
// ===== library types =====

// folder: AWCModbus/Modbus Services

TYPE "typeMasterData"
VERSION : 0.1
   STRUCT
      Done : Bool;   // Request Completed
      Busy : Bool;   // Modbus Service is Busy
      Error : Bool;   // Request returned error
      locked : Bool;   // internal mutex **DO NOT WRITE TO**
      Mode : USInt;   // internal mode **DO NOTE WRITE TO**
      Status : Int;   // Request Status
      "Slave ID" : UInt;   // internal slave ID **DO NOTE WRITE TO**
      "Register Address" : UDInt;   // internal register address **DO NOTE WRITE TO**
      Length : UInt;   // internal length **DO NOTE WRITE TO**
      RequestID : UInt;   // Request ID **DO NOTE WRITE TO**
      Data : Array[0..299] of Byte;   // Returned Data **DO NOTE WRITE TO**
   END_STRUCT;
END_TYPE

// folder: AWCModbus/01_Modbus Services

FUNCTION_BLOCK "ModbusRtuEngine"   // FB6, LAD
TITLE = ModbusRTUEngine
{ S7_Optimized_Access := 'TRUE' }
AUTHOR : Matt_Paulissen
FAMILY : AWCModbus
NAME : ModbusRTUEngine
// Modbus polling service for RTU devices.
   VAR_INPUT
      port : Port;   // The port references the “HW_Address” of the interface that will be used for Modbus communication. In the above example the “Local~CB_1241_(RS485) is referenced.
      baudRate : UDInt;   // The baud rate determines the communications speed of the network. All devices on the network must be set to the same baud rate. Available options are: 300, 600, 1200, 2400, 4800, 9600, 19200, 38400, 57600, 76800, 115200 bit/s.
      parity : UInt;   // Used to set the network parity. All devices on the network must have the same parity setting. Available options are: 0 = None, 1 = Odd, 2= Even.
      FirstScan : Bool;   // First Scan is used to initialize the communications port on system start up. This input can also be used at other times if it is desired to reset the communications parameters without restarting the CPU.
      Reset : Bool;   // Used to reinitialize the communications port of the CPU or module.
   END_VAR
   VAR_OUTPUT
      Status : Int;   // Returns any error code for the Modus Master function.
   END_VAR
   VAR_IN_OUT
      masterInterface : "typeMasterData";   // The “Master Interface” parameter is used to pass date between the Modbus RTU Engine and subsequent read and write function. The data type is the user defined type “typeMasterData”. It is necessary to create a global data block containing one instance of the “typeMasterData”.
   END_VAR
   VAR
      statPrevious : Int;
      statCurrent : Int;
      statIndex : Int;
      statRequestID : UInt;
      Comm_Load_Status : Int;
      Comm_Load_Done : Bool;
      Comm_Load_Error : Bool;
      instStuckInterfaceTimer : TON_TIME;
      instReinitilizeTimer : TON_TIME;
      instCommLoad : Modbus_Comm_Load;
      instMaster : Modbus_Master;
      inst7002Timeout : TON_TIME;
   END_VAR
   VAR_TEMP
      tempServerStatus : Int;
   END_VAR
   VAR CONSTANT
      UNITIALIZED : Int := 0;
      INITIALIZING_PORT : Int := 1;
      POLLING : Int := 2;
      POLLING_DONE : Int := 3;
   END_VAR
   VAR_TEMP   // added for the SCL form of the ladder/FBD networks
      _w1 : Bool;
   END_VAR
BEGIN

REGION Network 1: BLOCK INFO HEADER
   // AWC INC / (c)Copyright 2022
   // ------------------------------------------------------------------------------
   // Title:            ModbusRTUEngine_xxx
   // Comment/Function: Modbus Polling Service for RTU Devices:
   // Library/Family:   AWCModbus
   // Author:           Matt Paulissen
   // Tested with:      ---
   // Engineering:      TIA Portal V17
   // Restrictions:     -
   // Requirements:     ---
   // ------------------------------------------------------------------------------
   // Change log table:
   // Version  | Date       | Expert in charge       | Changes applied
   // ---------|------------|------------------------|------------------------------
   // 01.00.00 | 06.18.2018 | F.Maynard, M.Paulissen
   //                                Initial Release
   // 01.01.00 | 01.25.2019 | F.Maynard, M.Paulissen
   //                                Changed to RTU block that works for 1500 as well as 1200.
   // 02.00.00 | 03.12.2019 | F.Maynard, M.Paulissen
   //                                Changed all blocks to Optimized data access and added software unit.
   // 02.01.00 | 09.01.2019 | F.Maynard, M.Paulissen
   //                                Updated RTU engine to V4.3 instructions
   // 02.02.00 | 09.25.2019 | F.Maynard, M.Paulissen
   //                                Added remote TCP port for the TCP engine
   // 02.03.00 | 10.14.2019 | F.Maynard, M.Paulissen
   //                                 Bugfix for CM_PTP lockup
END_REGION

REGION Network 2: DESCRIPTION
   // The “ModbusRTUEngine” is used to communicate via Modbus RTU via an RS-485, RS-422, or RS-232 communications add on module.  The parameters are used to initialize the communication port, set the baud rate, and parity.
   // 
   // ---
   // 
   // CAUTION
   // :    You must change the mode parameter in instCommLoad to the correct value for your serial module
   // 
   // ---
END_REGION

REGION Network 3: Run Comm Load
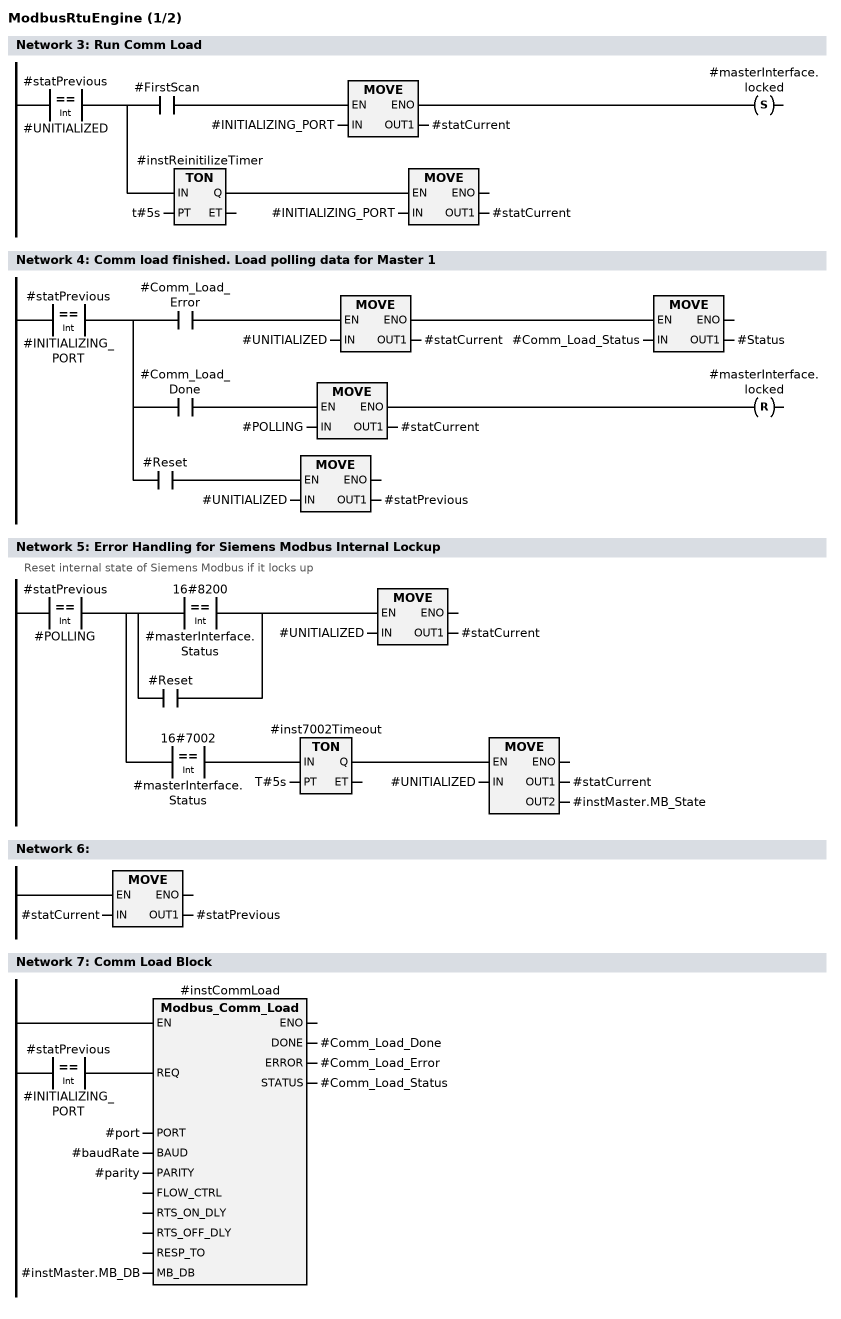
   #_w1 := #statPrevious = #UNITIALIZED;
   IF #_w1 AND #FirstScan THEN
       #statCurrent := #INITIALIZING_PORT;
       #masterInterface.locked := TRUE;
   END_IF;
   #instReinitilizeTimer(IN := #_w1, PT := t#5s);   // TON
   IF #instReinitilizeTimer.Q THEN #statCurrent := #INITIALIZING_PORT; END_IF;
END_REGION

REGION Network 4: Comm load finished. Load polling data for Master 1
   RUNG wire#powerrail
      { S7_Templates := "SrcType := Int" } EQ_Contact(in1 := #statPrevious, in2 := #INITIALIZING_PORT)
      wire#w1
      Contact( #Comm_Load_Error )
      Move(in := #UNITIALIZED, out1 => #statCurrent)
      Move(in := #Comm_Load_Status, out1 => #Status)
   END_RUNG
   RUNG wire#w1
      Contact( #Comm_Load_Done )
      Move(in := #POLLING, out1 => #statCurrent)
      R_Coil( #masterInterface.locked )
   END_RUNG
   RUNG wire#w1
      Contact( #Reset )
      Move(in := #UNITIALIZED, out1 => #statPrevious)
   END_RUNG
   // the same network as SCL:
   #_w1 := #statPrevious = #INITIALIZING_PORT;
   IF #_w1 AND #Comm_Load_Error THEN
       #statCurrent := #UNITIALIZED;
       #Status := #Comm_Load_Status;
   END_IF;
   IF #_w1 AND #Comm_Load_Done THEN
       #statCurrent := #POLLING;
       #masterInterface.locked := FALSE;
   END_IF;
   IF #_w1 AND #Reset THEN #statPrevious := #UNITIALIZED; END_IF;
END_REGION

REGION Network 5: Error Handling for Siemens Modbus Internal Lockup
   // Reset internal state of Siemens Modbus if it locks up
   #_w1 := #statPrevious = #POLLING;
   IF #_w1 AND ((16#8200 = #masterInterface.Status) OR #Reset) THEN #statCurrent := #UNITIALIZED; END_IF;
   #inst7002Timeout(IN := #_w1 AND (16#7002 = #masterInterface.Status), PT := T#5s);   // TON
   IF #inst7002Timeout.Q THEN
       #statCurrent := #UNITIALIZED;
       #instMaster.MB_State := #UNITIALIZED;
   END_IF;
END_REGION

REGION Network 6
   RUNG wire#powerrail
      Move(in := #statCurrent, out1 => #statPrevious)
   END_RUNG
   // the same network as SCL:
   #statPrevious := #statCurrent;
END_REGION

REGION Network 7: Comm Load Block
   #instCommLoad(REQ := #statPrevious = #INITIALIZING_PORT,   // Modbus_Comm_Load
                 PORT := #port,
                 BAUD := #baudRate,
                 PARITY := #parity,
                 MB_DB := #instMaster.MB_DB,
                 DONE => #Comm_Load_Done,
                 ERROR => #Comm_Load_Error,
                 STATUS => #Comm_Load_Status);
END_REGION

REGION Network 8: Master Instance 1
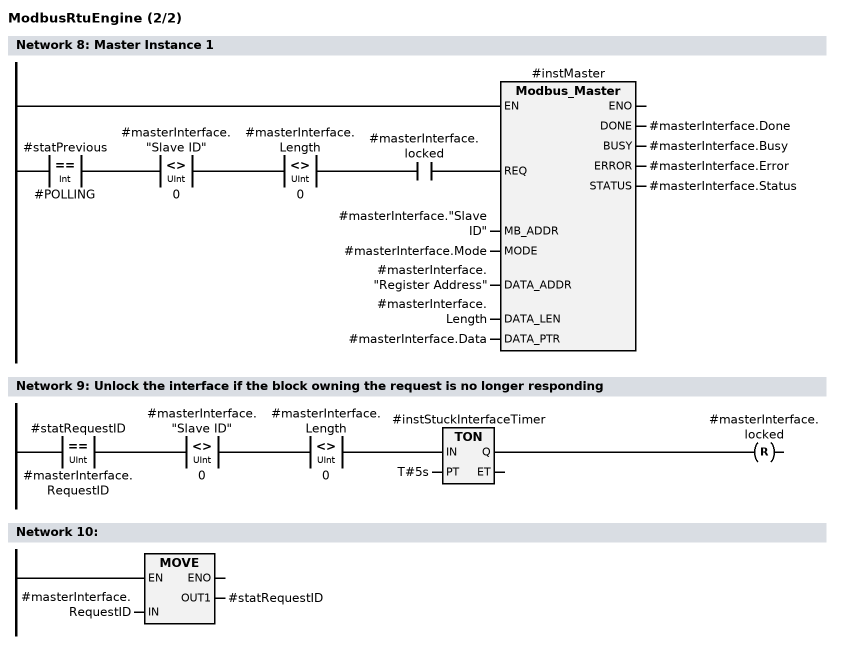
   #instMaster(REQ := (#statPrevious = #POLLING) AND (#masterInterface."Slave ID" <> 0) AND (#masterInterface.Length <> 0) AND #masterInterface.locked,   // Modbus_Master
               MB_ADDR := #masterInterface."Slave ID",
               MODE := #masterInterface.Mode,
               DATA_ADDR := #masterInterface."Register Address",
               DATA_LEN := #masterInterface.Length,
               DATA_PTR := #masterInterface.Data,
               DONE => #masterInterface.Done,
               BUSY => #masterInterface.Busy,
               ERROR => #masterInterface.Error,
               STATUS => #masterInterface.Status);
END_REGION

REGION Network 9: Unlock the interface if the block owning the request is no longer responding
   #instStuckInterfaceTimer(IN := (#statRequestID = #masterInterface.RequestID) AND (#masterInterface."Slave ID" <> 0) AND (#masterInterface.Length <> 0),   // TON
                           PT := T#5s);
   IF #instStuckInterfaceTimer.Q THEN #masterInterface.locked := FALSE; END_IF;
END_REGION

REGION Network 10
   RUNG wire#powerrail
      Move(in := #masterInterface.RequestID, out1 => #statRequestID)
   END_RUNG
   // the same network as SCL:
   #statRequestID := #masterInterface.RequestID;
END_REGION
END_FUNCTION_BLOCK

FUNCTION_BLOCK "ModbusTCPEngine"   // FB22, LAD
TITLE = ModbusTCPEngine
{ S7_Optimized_Access := 'TRUE' }
AUTHOR : Matt_Paulissen
FAMILY : AWCModbus
NAME : ModbusTCPEngine
VERSION : 0.1
// The “ModbusTCPEngine” is used to communicate via Modbus TCP via the on-board Profinet port or via a separate add on Ethernet communications module.
   VAR_INPUT
      port : Hw_Any;   // The port references the “HW_Address” of the Profinet interface that will be used for Modbus TCP communication. In the above example the “Local~Profinet_interface_1” is referenced.
      connectionId : Conn_Ouc;   // Defines the unique connection id for the Modbus Client. If more than one instance of the Modbus Client is used a different connection id must be assigned.
      tcpPort : UInt;   // Modbus TCP Server TCP Port Number. Typically this is port 502, but in some instances may be changed to meet network requirements.
      ipOne : Byte;   // First address octet of the server to be polled.
      ipTwo : Byte;   // Second address octet of the server to be polled.
      ipThree : Byte;   // Third address octet of the server to be polled.
      ipFour : Byte;   // Fourth address octet of the server to be polled.
   END_VAR
   VAR_OUTPUT
      Status : Int;   // Returns any error code for the Modbus Client function.
   END_VAR
   VAR_IN_OUT
      masterInterface : "typeMasterData";   // The “Master Interface” parameter is used to pass date between the Modbus RTU Engine and subsequent read and write function. The data type is the user defined type “typeMasterData”. It is necessary to create a global data block containing one instance of the “typeMasterData”.
   END_VAR
   VAR
      instClient : MB_CLIENT;
      connection : TCON_IP_v4;
      statRequestID : UInt;
      instStuckInterfaceTimer : TON_TIME;
   END_VAR
   VAR CONSTANT
      UNITIALIZED : Int := 0;
      INITIALIZING_PORT : Int := 1;
      POLLING_ONE : Int := 2;
      POLLING_DONE_ONE : Int := 3;
      POLLING_TWO : Int := 4;
      POLLING_TWO_DONE : Int := 5;
   END_VAR
   // connection.ConnectionType := 11;
   // connection.ActiveEstablished := 1;
   // connection.RemotePort := 502;
   // connection.LocalPort := 502;
BEGIN

REGION Network 1: BLOCK INFO HEADER
   // AWC INC / (c)Copyright 2022
   // ------------------------------------------------------------------------------
   // Title:            ModbusTCPEngine_xxx
   // Comment/Function: Modbus Polling Service for RTU Devices:
   // Library/Family:   AWCModbus
   // Author:           Matt Paulissen
   // Tested with:      ---
   // Engineering:      TIA Portal V17
   // Restrictions:     -
   // Requirements:     ---
   // ------------------------------------------------------------------------------
   // Change log table:
   // Version  | Date       | Expert in charge       | Changes applied
   // ---------|------------|------------------------|------------------------------
   // 01.00.00 | 06.18.2018 | F.Maynard, M.Paulissen | Initial Release
   // 01.01.00 | 01.25.2019 | F.Maynard, M.Paulissen | Changed to RTU block that works for 1500 as well as 1200.  Added Devices folder for common devices.  Added ability to read from contacts and write to coils with Boolean tags
   // 02.00.00 | 03.12.2019 | F.Maynard, M.Paulissen | Changed all blocks to Optimized data access and added software unit.
   // 02.01.00 | 09.01.2019 | F.Maynard, M.Paulissen | Updated RTU engine to V4.3 instructions
   // 02.02.00 | 09.25.2019 | F.Maynard, M.Paulissen | Added remote TCP port for the TCP engine
   // 02.03.00 | 10.14.2019 | F.Maynard, M.Paulissen | Bugfix for CM_PTP lockup
END_REGION

REGION Network 2: DESCRIPTION
   // The “ModbusTCPEngine” is used to communicate via Modbus TCP via the on-board Profinet port or via a separate add on Ethernet communications module.
END_REGION

REGION Network 3: Move ip address from interface to static tcon_ip_v4
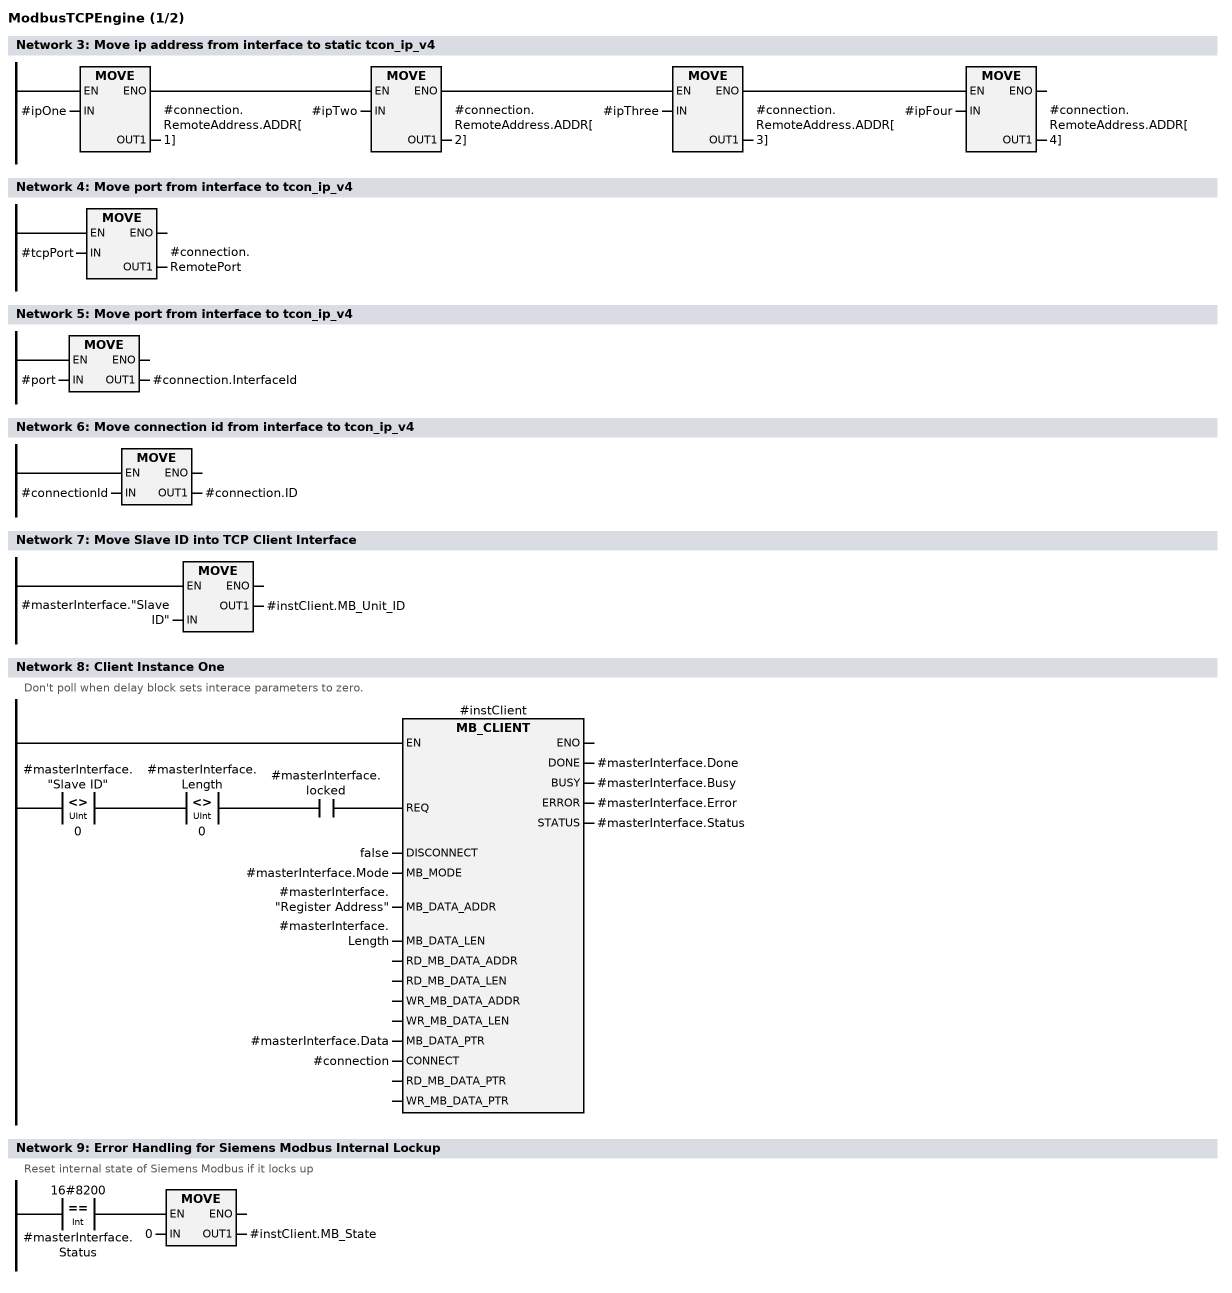
   RUNG wire#powerrail
      Move(in := #ipOne, out1 => #connection.RemoteAddress.ADDR[1])
      Move(in := #ipTwo, out1 => #connection.RemoteAddress.ADDR[2])
      Move(in := #ipThree, out1 => #connection.RemoteAddress.ADDR[3])
      Move(in := #ipFour, out1 => #connection.RemoteAddress.ADDR[4])
   END_RUNG
   // the same network as SCL:
   #connection.RemoteAddress.ADDR[1] := #ipOne;
   #connection.RemoteAddress.ADDR[2] := #ipTwo;
   #connection.RemoteAddress.ADDR[3] := #ipThree;
   #connection.RemoteAddress.ADDR[4] := #ipFour;
END_REGION

REGION Network 4: Move port from interface to tcon_ip_v4
   RUNG wire#powerrail
      Move(in := #tcpPort, out1 => #connection.RemotePort)
   END_RUNG
   // the same network as SCL:
   #connection.RemotePort := #tcpPort;
END_REGION

REGION Network 5: Move port from interface to tcon_ip_v4
   RUNG wire#powerrail
      Move(in := #port, out1 => #connection.InterfaceId)
   END_RUNG
   // the same network as SCL:
   #connection.InterfaceId := #port;
END_REGION

REGION Network 6: Move connection id from interface to tcon_ip_v4
   RUNG wire#powerrail
      Move(in := #connectionId, out1 => #connection.ID)
   END_RUNG
   // the same network as SCL:
   #connection.ID := #connectionId;
END_REGION

REGION Network 7: Move Slave ID into TCP Client Interface
   RUNG wire#powerrail
      Move(in := #masterInterface."Slave ID", out1 => #instClient.MB_Unit_ID)
   END_RUNG
   // the same network as SCL:
   #instClient.MB_Unit_ID := #masterInterface."Slave ID";
END_REGION

REGION Network 8: Client Instance One
   // Don't poll when delay block sets interace parameters to zero.
   #instClient(REQ := (#masterInterface."Slave ID" <> 0) AND (#masterInterface.Length <> 0) AND #masterInterface.locked,   // MB_CLIENT
               DISCONNECT := false,
               MB_MODE := #masterInterface.Mode,
               MB_DATA_ADDR := #masterInterface."Register Address",
               MB_DATA_LEN := #masterInterface.Length,
               MB_DATA_PTR := #masterInterface.Data,
               CONNECT := #connection,
               DONE => #masterInterface.Done,
               BUSY => #masterInterface.Busy,
               ERROR => #masterInterface.Error,
               STATUS => #masterInterface.Status);
END_REGION

REGION Network 9: Error Handling for Siemens Modbus Internal Lockup
   // Reset internal state of Siemens Modbus if it locks up
   RUNG wire#powerrail
      { S7_Templates := "SrcType := Int" } EQ_Contact(in1 := 16#8200, in2 := #masterInterface.Status)
      Move(in := 0, out1 => #instClient.MB_State)
   END_RUNG
   // the same network as SCL:
   IF 16#8200 = #masterInterface.Status THEN #instClient.MB_State := 0; END_IF;
END_REGION

REGION Network 10: Unlock the interface if the block owning the request is no longer responding
   // Modbus Polling Delay block sets interfaces to zero.  Don't want to unlock interface if this block is holding it.
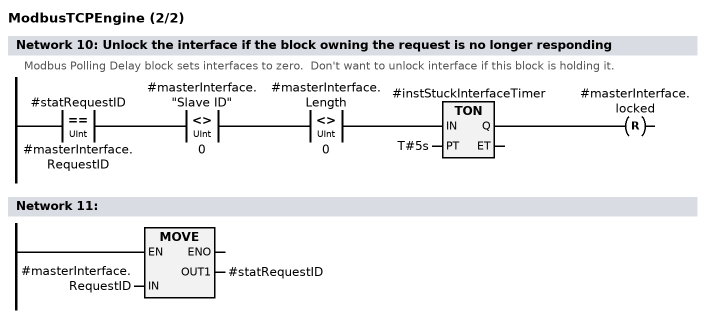
   #instStuckInterfaceTimer(IN := (#statRequestID = #masterInterface.RequestID) AND (#masterInterface."Slave ID" <> 0) AND (#masterInterface.Length <> 0),   // TON
                           PT := T#5s);
   IF #instStuckInterfaceTimer.Q THEN #masterInterface.locked := FALSE; END_IF;
END_REGION

REGION Network 11
   RUNG wire#powerrail
      Move(in := #masterInterface.RequestID, out1 => #statRequestID)
   END_RUNG
   // the same network as SCL:
   #statRequestID := #masterInterface.RequestID;
END_REGION
END_FUNCTION_BLOCK

// folder: AWCModbus/01_Modbus Services/Modbus Polling Functions

FUNCTION "GeneralModbusPoll" : Void   // FC11, SCL
TITLE = GeneralModbusPoll
{ S7_Optimized_Access := 'TRUE' }
AUTHOR : Matt_Paulissen
FAMILY : AWCModbus
NAME : GeneralModbusPoll
VERSION : 0.1
// The General Modbus Poll Function is used to read a single data value from the Modbus RTU slave or Modbus TCP server.
   VAR_INPUT
      slaveId : Int;   // When using the function for Modbus RTU this will be the remote slave network address. When using the function for Modbus TCP this will be the device address, in most instances this value will be 1, unless there is a Modbus TCP to Modbus RTU gateway employed. If there is a Modbus TCP to Modbus RTU gateway this value will point to the slave device address on the Modbus RTU side of the gateway.
      address : UDInt;   // The address parameter references the Modbus register that will be polled.
      swappedFloatingPoint : Bool;   // When reading floating point values from some devices it is necessary to reverse the order of the received data words to display the value correctly. In this it is necessary to set this value to True.
      substituteValue : Real;   // If the remote device fails to respond or has an error the Substitute Value will be returned to the Data value. This can be used to alert the operator that there is a problem with the connection.
   END_VAR
   VAR_OUTPUT
      data : Variant;   // The Data parameter is the value returned from the device. The data type of the PLC variable selected will determine how many registers are requested from the device and how they are displayed in the PLC.
   END_VAR
   VAR_IN_OUT
      modbusInterface : "typeMasterData";   // The “Master Interface” parameter is used to pass date between the Modbus RTU Engine and subsequent read and write function. The data type is the user defined type “typeMasterData”. It is necessary to create a global data block containing one instance of the “typeMasterData”.
   END_VAR
   VAR_TEMP
      tempArray : Array[0..3] of Byte;
      tempDWord : DWord;
      tempStatus : Int;
      tempPos : DInt;
      tempBool : Bool;
   END_VAR
BEGIN
   REGION BLOCK INFO HEADER
       //===============================================================================
       // AWC INC / (c)Copyright 2022
       //-------------------------------------------------------------------------------
       // Title:            GeneralModbusPoll_xxx
       // Comment/Function: Poll an individual value from a Modbus Device
       // Library/Family:   AWCModbus
       // Author:           Matt Paulissen
       // Tested with:      ---
       // Engineering:      TIA Portal V17
       // Restrictions:     ---
       // Requirements:     ---
       //-------------------------------------------------------------------------------
       // Change log table:
       // Version  | Date       | Expert in charge       | Changes applied
       //----------|------------|------------------------|------------------------------
       // 01.00.00 | 08.09.2017 | Matt Paulissen | First released version
       // 01.00.01 | 08.23.2017 | Matt Paulissen | Added ability to set failover value
       // 01.00.02 | 09.21.2018 | Matt Paulissen | Added request ID to detect stuck lock
       // 01.01.00 | 01.25.2019 | Matt Paulissen | Added ability to read contacts
       // 01.01.01 | 11.04.2022 | Matt Paulissen | Bug fix for substitute value on DWord
       //===============================================================================
   END_REGION

   REGION DESCRIPTION
       (/*The General Modbus Poll Function is used to read a single data value from the Modbus RTU slave or Modbus TCP server.*/)
   END_REGION DESCRIPTION

   //Check for lock
   IF (NOT #modbusInterface.locked) THEN
       //Move Register and Slave address to Modbus Register
       #modbusInterface."Slave ID" := #slaveId;
       #modbusInterface."Register Address" := #address;
       #modbusInterface.Mode := 0;
       CASE TypeOf(#data) OF
           UInt:
               #modbusInterface.Length := 1;
           Int:
               #modbusInterface.Length := 1;
           Word:
               #modbusInterface.Length := 1;
           DWord:
               #modbusInterface.Length := 2;
           Real:
               #modbusInterface.Length := 2;
           Bool:
               #modbusInterface.Length := 1;
           ELSE  // Statement section ELSE
               ;
       END_CASE;
       #modbusInterface.locked := TRUE;
       #modbusInterface.RequestID += 1;
       RETURN;
   END_IF;
   IF ((#modbusInterface.locked)
       AND (
       (#modbusInterface."Slave ID" = #slaveId)
       AND (#modbusInterface."Register Address" = #address)
       AND (#modbusInterface.Mode = 0))
       )
   THEN
       IF (#modbusInterface.Done) THEN
           //Inspect type of output and set correct type of input in modbus register
           CASE TypeOf(#data) OF
               UInt:
                   #tempStatus := Deserialize(SRC_ARRAY := #modbusInterface.Data,
                                              DEST_VARIABLE => #data,
                                              POS := #tempPos);
               Int:
                   #tempStatus := Deserialize(SRC_ARRAY := #modbusInterface.Data,
                                              DEST_VARIABLE => #data,
                                              POS := #tempPos);
               Word:
                   #tempStatus := Deserialize(SRC_ARRAY := #modbusInterface.Data,
                                              DEST_VARIABLE => #data,
                                              POS := #tempPos);
               DWord:
                   IF #swappedFloatingPoint THEN
                       // Swapped 
                       #tempArray[3] := #modbusInterface.Data[1];
                       #tempArray[2] := #modbusInterface.Data[0];
                       #tempArray[1] := #modbusInterface.Data[3];
                       #tempArray[0] := #modbusInterface.Data[2];
                       #tempStatus := Deserialize(SRC_ARRAY := #tempArray,
                                                  DEST_VARIABLE => #data,
                                                  POS := #tempPos);
                   ELSE
                       //Consecutive
                       #tempStatus := Deserialize(SRC_ARRAY := #modbusInterface.Data,
                                                  DEST_VARIABLE => #data,
                                                  POS := #tempPos);
                   END_IF;

               Real:
                   IF #swappedFloatingPoint THEN
                       // Swapped 
                       #tempArray[3] := #modbusInterface.Data[1];
                       #tempArray[2] := #modbusInterface.Data[0];
                       #tempArray[1] := #modbusInterface.Data[3];
                       #tempArray[0] := #modbusInterface.Data[2];
                       #tempStatus := Deserialize(SRC_ARRAY := #tempArray,
                                                  DEST_VARIABLE => #data,
                                                  POS := #tempPos);

                   ELSE
                       //Consecutive
                       #tempStatus := Deserialize(SRC_ARRAY := #modbusInterface.Data,
                                                  DEST_VARIABLE => #data,
                                                  POS := #tempPos);
                   END_IF;

               Bool:
                   #tempBool := #modbusInterface.Data[0].%X0;
                   VariantPut(SRC := #tempBool,
                              DST := #data);
               ELSE  // Statement section ELSE
                   ;
           END_CASE;
           #modbusInterface.locked := FALSE;
       END_IF;
       IF (#modbusInterface.Error) THEN
           CASE TypeOf(#data) OF
               UInt:
                   VariantPut(SRC := REAL_TO_UINT(IN:=#substituteValue),
                              DST := #data);
               Int:
                   VariantPut(SRC := REAL_TO_INT(IN := #substituteValue),
                              DST := #data);
               Word:
                   VariantPut(SRC := INT_TO_WORD(IN:=TRUNC_INT(IN := #substituteValue)),
                              DST := #data);
               DWord:
                   VariantPut(SRC := REAL_TO_DWORD(IN:=#substituteValue),
                              DST := #data);
               Real:
                   VariantPut(SRC := #substituteValue,
                              DST := #data);
               Bool:
                   IF (#substituteValue <> 0.0) THEN
                       #tempBool := TRUE;
                   ELSE
                       #tempBool := FALSE;
                   END_IF;
                   VariantPut(SRC := #tempBool,
                              DST := #data);
               ELSE  // Statement section ELSE
                   ;
           END_CASE;
           #modbusInterface.locked := 0;
       END_IF;
   END_IF;
END_FUNCTION

FUNCTION "LargeModbusPoll" : Void   // FC892, SCL
TITLE = LargeModbusPoll
{ S7_Optimized_Access := 'TRUE' }
AUTHOR : Matt_Paulissen
FAMILY : AWCModbus
NAME : LargeModbusPoll
VERSION : 0.1
// Large Modbus Poll function is used to read multiple contiguous data values from a Modbus RTU slave or Modbus TCP Server. Number of values read is determined by the size of the Array element at the Data parameter.
   VAR_INPUT
      slaveId : Int;   // When using the function for Modbus RTU this will be the remote slave network address. When using the function for Modbus TCP this will be the device address, in most instances this value will be 1, unless there is a Modbus TCP to Modbus RTU gateway employed. If there is a Modbus TCP to Modbus RTU gateway this value will point to the slave device address on the Modbus RTU side of the gateway.
      address : UDInt;   // The address parameter references the Modbus register that will be polled.
   END_VAR
   VAR_OUTPUT
      data : Variant;   // The Data parameter is the value returned from the device. The data type of the PLC variable selected will determine how many registers are requested from the device and how they are displayed in the PLC. The allowable data types are: Int, UInt, Word, Dint, UDint, DWord, and Real, Array of Uint, Array of Int, Array of Udint, Array of Dint, Array of Real, and PLC UDTs. Care should be taken to not exceed the 127-byte limitation of the Modbus Read Function.
      status : Int;   // Returns any error code for the Modbus Master function.
   END_VAR
   VAR_IN_OUT
      modbusInterface : "typeMasterData";   // The “Master Interface” parameter is used to pass datae between the Modbus RTU Engine and subsequent read and write function. The data type is the user defined type “typeMasterData”. It is necessary to create a global data block containing one instance of the “typeMasterData”.
   END_VAR
   VAR_TEMP
      tempPosition : DInt;
      tempStatus : Int;
      tempMode : USInt;
      tempAddress : UInt;
   END_VAR
BEGIN
   REGION BLOCK INFO HEADER
       //===============================================================================
       // AWC INC / (c)Copyright 2022
       //-------------------------------------------------------------------------------
       // Title:            LargeModbusPoll_xxx
       // Comment/Function: Read multiple contiguous values from a Modbus Device
       // Library/Family:   AWCModbus
       // Author:           Matt Paulissen
       // Tested with:      ---
       // Engineering:      TIA Portal V17
       // Restrictions:     ---
       // Requirements:     ---
       //-------------------------------------------------------------------------------
       // Change log table:
       // Version  | Date       | Expert in charge       | Changes applied
       //----------|------------|------------------------|------------------------------
       // 01.00.00 | 05.17.2018 | Matt Paulissen | First released version
       // 01.00.02 | 09.21.2018 | Matt Paulissen | Added request ID to detect stuck lock
       // 01.01.06 | 09.29.2020 | Matt Paulissen | Added extended modbus addressing
       // 01.01.07 | 11.16.2022 | Matt Paulissen | Allowed UDint for addresses
       //===============================================================================
   END_REGION

   REGION DESCRIPTION
       (/*Large Modbus Poll function is used to read multiple contiguous data values from a Modbus RTU slave or Modbus TCP Server.
       Number of values read is determined by the size of the Array element at the Data parameter.*/)
   END_REGION DESCRIPTION

   //Check for lock
   IF (NOT #modbusInterface.locked) THEN
       //Move Register and Slave address to Modbus Register
       #modbusInterface."Slave ID" := #slaveId;
       #modbusInterface."Register Address" := #address;

       //Get UDT length in bytes
       #tempStatus := Serialize(SRC_VARIABLE := #data, DEST_ARRAY => #modbusInterface.Data, POS := #tempPosition);
       IF (#tempStatus <> 0) THEN  //Exit instruction if UDT cannot be processed by the modbus interface
           RETURN;
       END_IF;
       //Get number of registers needed to poll entire UDT
       CASE #address OF
           1..9999, 10001..19999:  //Edge case for boolean values
               #tempPosition := #tempPosition * 8; //Multiply bytes by 8 to get bits
           50000..59999:  //Edge case for extended addressing
               #modbusInterface.Mode := 104;
               #modbusInterface."Register Address" := #address - 40001;
               IF ((#tempPosition MOD 2) = 0) THEN
                   #tempPosition := #tempPosition / 2;
               ELSE
                   #tempPosition := (#tempPosition / 2) + 1;
               END_IF;
           ELSE  //Normal registers
               #modbusInterface.Mode := 0;
               IF ((#tempPosition MOD 2) = 0) THEN
                   #tempPosition := #tempPosition / 2;
               ELSE
                   #tempPosition := (#tempPosition / 2) + 1;
               END_IF;
       END_CASE;
       #modbusInterface.Length := #tempPosition;
       #modbusInterface.locked := TRUE;
       #modbusInterface.RequestID += 1;
       RETURN;
   END_IF;
   //Edge case handling for extended modbus addressing
   IF (#address >= 50000 AND #address <= 59999) THEN
       #tempAddress := #address - 40001;
       #tempMode := 104;
   ELSE
       #tempAddress := #address;
       #tempMode := 0;
   END_IF;
   IF ((#modbusInterface.locked)
       AND (
       (#modbusInterface."Slave ID" = #slaveId)
       AND (#modbusInterface."Register Address" = #tempAddress)
       AND (#modbusInterface.Mode = #tempMode))
       )
   THEN
       IF (#modbusInterface.Done) THEN
           //Deserialize to output
           #tempStatus := Deserialize(SRC_ARRAY := #modbusInterface.Data, DEST_VARIABLE => #data, POS := #tempPosition);
           #modbusInterface.locked := FALSE;
           #status := #modbusInterface.Status;
       END_IF;
       IF (#modbusInterface.Error) THEN
           //TODO: error handling for variant????
           #modbusInterface.locked := 0;
           #status := #modbusInterface.Status;
       END_IF;
   END_IF;
END_FUNCTION

FUNCTION "GeneralModbusWrite" : Void   // FC893, SCL
TITLE = GeneralModbusWrite
{ S7_Optimized_Access := 'TRUE' }
AUTHOR : Matt_Paulissen
FAMILY : AWCModbus
NAME : GeneralModbusWrite
VERSION : 0.1
// The data to be written to the remote device.
   VAR_INPUT
      slaveId : Int;   // When using the function for Modbus RTU this will be the remote slave network address. When using the function for Modbus TCP this will be the device address, in most instances this value will be 1, unless there is a Modbus TCP to Modbus RTU gateway employed. If there is a Modbus TCP to Modbus RTU gateway this value will point to the slave device address on the Modbus RTU side of the gateway.
      address : UDInt;   // The address parameter references the Modbus register that will be written.
      write : Bool;   // Data will be written to the remote device as long as this is set to TRUE.
      data : Variant;   // The data to be written to the remote device.
      swappedFloatingPoint : Bool;   // When writing floating point values to some devices it is necessary to reverse the order of the sent data words to display the value correctly. In this it is necessary to set this value to True.
   END_VAR
   VAR_OUTPUT
      status : Word;   // Returns any error code for the Modbus Master function.
   END_VAR
   VAR_IN_OUT
      modbusInterface : "typeMasterData";   // The “Master Interface” parameter is used to pass datae between the Modbus RTU Engine and subsequent read and write function. The data type is the user defined type “typeMasterData”. It is necessary to create a global data block containing one instance of the “typeMasterData”.
   END_VAR
   VAR_TEMP
      tempdWord : DWord;
      tempUint : UInt;
      tempInt : Int;
      tempWord : Word;
      tempReal : Real;
      tempBool : Bool;
      tempStatus : Int;
      tempPos : DInt;
   END_VAR
   VAR CONSTANT
      WRITE_OK : Word := 16#7000;
   END_VAR
BEGIN
   REGION BLOCK INFO HEADER
       //===============================================================================
       // AWC INC / (c)Copyright 2022
       //-------------------------------------------------------------------------------
       // Title:            GeneralModbusWrite_xxx
       // Comment/Function: Write an individual value from a Modbus Device
       // Library/Family:   AWCModbus
       // Author:           Matt Paulissen
       // Tested with:      ---
       // Engineering:      TIA Portal V17
       // Restrictions:     ---
       // Requirements:     ---
       //-------------------------------------------------------------------------------
       // Change log table:
       // Version  | Date       | Expert in charge       | Changes applied
       //----------|------------|------------------------|------------------------------
       // 01.00.00 | 08.09.2017 | Matt Paulissen | First released version
       // 01.00.01 | 08.23.2017 | Matt Paulissen | Added ability to set failover value
       // 01.00.02 | 09.21.2018 | Matt Paulissen | Added request ID to detect stuck lock
       // 01.01.00 | 01.25.2019 | Matt Paulissen | Added ability to read contacts
       // 01.01.07 | 03.16.2021 | Matt Paulissen | Bug Fix for writing single coil
       // 01.01.08 | 11.16.2022 | Matt Paulissen | Allowed UDint for Addresses
       //===============================================================================
   END_REGION

   REGION DESCRIPTION
       (/*The General Modbus Write function is used to write a single data value to a Modbus RTU Slave or Modbus TCP Server.*/)
   END_REGION DESCRIPTION

   //Check for lock
   IF ((NOT #modbusInterface.locked) AND (#write)) THEN
       //Move Register and Slave address to Modbus Register
       #modbusInterface."Slave ID" := #slaveId;
       #modbusInterface."Register Address" := #address;
       #modbusInterface.Mode := 1;
       CASE TypeOf(#data) OF
           UInt:
               #modbusInterface.Length := 1;
               //VariantGet(SRC:=#data,
               //           DST=>#tempUint);
               #tempStatus := Serialize(SRC_VARIABLE := #data, DEST_ARRAY => #modbusInterface.Data, POS := #tempPos);

               //#modbusInterface.Data[0] := #tempUint;
           Int:
               #modbusInterface.Length := 1;
               // VariantGet(SRC := #data,
               //            DST => #tempInt);
               // #modbusInterface.Data[0] := INT_TO_UINT(IN:=#tempInt);
               #tempStatus := Serialize(SRC_VARIABLE := #data, DEST_ARRAY => #modbusInterface.Data, POS := #tempPos);
           Word:
               #modbusInterface.Length := 1;
               // VariantGet(SRC := #data,
               //            DST => #tempWord);
               // #modbusInterface.Data[0] := WORD_TO_UINT(IN := #tempWord);
               #tempStatus := Serialize(SRC_VARIABLE := #data, DEST_ARRAY => #modbusInterface.Data, POS := #tempPos);
           DWord:
               #modbusInterface.Length := 2;
               VariantGet(SRC := #data,
                          DST => #tempdWord);
               IF #swappedFloatingPoint THEN
                   // Swapped 
                   #modbusInterface.Data[2] := #tempdWord.%B3;
                   #modbusInterface.Data[3] := #tempdWord.%B2;
                   #modbusInterface.Data[0] := #tempdWord.%B1;
                   #modbusInterface.Data[1] := #tempdWord.%B0;
               ELSE
                   //Consecutive
                   #modbusInterface.Data[3] := #tempdWord.%B0;
                   #modbusInterface.Data[2] := #tempdWord.%B1;
                   #modbusInterface.Data[1] := #tempdWord.%B2;
                   #modbusInterface.Data[0] := #tempdWord.%B3;
               END_IF;
           Real:
               #modbusInterface.Length := 2;
               VariantGet(SRC := #data,
                          DST => #tempReal);
               #tempdWord := REAL_TO_DWORD(IN:=#tempReal);
               IF #swappedFloatingPoint THEN
                   // Swapped 
                   #modbusInterface.Data[2] := #tempdWord.%B3;
                   #modbusInterface.Data[3] := #tempdWord.%B2;
                   #modbusInterface.Data[0] := #tempdWord.%B1;
                   #modbusInterface.Data[1] := #tempdWord.%B0;
               ELSE
                   //Consecutive
                   #modbusInterface.Data[3] := #tempdWord.%B0;
                   #modbusInterface.Data[2] := #tempdWord.%B1;
                   #modbusInterface.Data[1] := #tempdWord.%B2;
                   #modbusInterface.Data[0] := #tempdWord.%B3;
               END_IF;
           Bool:
               #modbusInterface.Length := 1;
               VariantGet(SRC := #data,
                          DST => #tempBool);
               // Cleared buffer to fix bug during single coil writes
               #modbusInterface.Data[0] := 0;
               #modbusInterface.Data[1] := 0;
               #modbusInterface.Data[0].%X0 := #tempBool;
           ELSE  // Statement section ELSE
               ;
       END_CASE;
       #modbusInterface.locked := TRUE;
       #modbusInterface.RequestID += 1;
       RETURN;
   END_IF;
   IF ((#modbusInterface.locked)
       AND (
       (#modbusInterface."Slave ID" = #slaveId)
       AND (#modbusInterface."Register Address" = #address)
       AND (#modbusInterface.Mode = 1))
       )
   THEN
       IF (#modbusInterface.Done) THEN
           //Inspect type of output and set correct type of input in modbus register
           #status := #WRITE_OK;
           #modbusInterface.locked := FALSE;
       END_IF;
       IF (#modbusInterface.Error) THEN
           #status := #modbusInterface.Status;
           #modbusInterface.locked := false;
       END_IF;
   END_IF;
END_FUNCTION

FUNCTION "LargeModbusWrite" : Void   // FC894, SCL
TITLE = LargeModbusWrite
{ S7_Optimized_Access := 'TRUE' }
AUTHOR : Matt_Paulissen
FAMILY : AWCModbus
NAME : LargeModbusWrite
VERSION : 0.1
// The General Modbus Write function is used to write a single data value to a Modbus RTU Slave or Modbus TCP Server.
   VAR_INPUT
      slaveId : Int;   // When using the function for Modbus RTU this will be the remote slave network address. When using the function for Modbus TCP this will be the device address, in most instances this value will be 1, unless there is a Modbus TCP to Modbus RTU gateway employed. If there is a Modbus TCP to Modbus RTU gateway this value will point to the slave device address on the Modbus RTU side of the gateway.
      address : UDInt;   // The address parameter references the Modbus register that will be written.
      write : Bool;   // Data will be written to the remote device as long as this is set to TRUE.
      data : Variant;   // The data to be written to the remote device.
   END_VAR
   VAR_OUTPUT
      status : Word;   // Returns any error code for the Modbus Master function.
   END_VAR
   VAR_IN_OUT
      modbusInterface : "typeMasterData";   // The “Master Interface” parameter is used to pass data between the Modbus RTU Engine and subsequent read and write function. The data type is the user defined type “typeMasterData”. It is necessary to create a global data block containing one instance of the “typeMasterData”.
   END_VAR
   VAR_TEMP
      tempPosition : DInt;
      tempStatus : Int;
   END_VAR
   VAR CONSTANT
      WRITE_OK : Word := 16#7000;
   END_VAR
BEGIN
   REGION BLOCK INFO HEADER
       //===============================================================================
       // AWC INC / (c)Copyright 2022
       //-------------------------------------------------------------------------------
       // Title:            LargeModbusPoll_xxx
       // Comment/Function: Write multiple contiguous values from a Modbus Device
       // Library/Family:   AWCModbus
       // Author:           Matt Paulissen
       // Tested with:      ---
       // Engineering:      TIA Portal V17
       // Restrictions:     ---
       // Requirements:     ---
       //-------------------------------------------------------------------------------
       // Change log table:
       // Version  | Date       | Expert in charge       | Changes applied
       //----------|------------|------------------------|------------------------------
       // 01.00.00 | 05.17.2018 | Matt Paulissen | First released version
       // 01.00.02 | 09.21.2018 | Matt Paulissen | Added request ID to detect stuck lock
       // 01.00.03 | 11.16.2022 | Matt Paulissen | Allowed UDint for Addresses
       //===============================================================================
   END_REGION

   REGION DESCRIPTION
       (/*The General Modbus Write function is used to write a single data value to a Modbus RTU Slave or Modbus TCP Server.*/)
   END_REGION DESCRIPTION

   //Check for lock
   IF ((NOT #modbusInterface.locked) AND (#write)) THEN
       //Move Register and Slave address to Modbus Register
       #modbusInterface."Slave ID" := #slaveId;
       #modbusInterface."Register Address" := #address;
       #modbusInterface.Mode := 1;
       //Move data to interface and get length
       #tempStatus := Serialize(SRC_VARIABLE := #data, DEST_ARRAY => #modbusInterface.Data, POS := #tempPosition);
       IF (#tempStatus <> 0) THEN  //Exit instruction if UDT cannot be processed by the modbus interface
           RETURN;
       END_IF;
       //Get number of registers needed to poll entire UDT
       CASE #address OF
           1..9999, 10001..19999:  //Edge case for boolean values
               #tempPosition := #tempPosition * 8; //Multiply bytes by 8 to get bits
           ELSE  //Normal registers
               IF ((#tempPosition MOD 2) = 0) THEN
                   #tempPosition := #tempPosition / 2;
               ELSE
                   #tempPosition := (#tempPosition / 2) + 1;
               END_IF;
       END_CASE;
       #modbusInterface.Length := #tempPosition;
       #modbusInterface.locked := TRUE;
       #modbusInterface.RequestID += 1;
       RETURN;
   END_IF;
   IF ((#modbusInterface.locked)
       AND (
       (#modbusInterface."Slave ID" = #slaveId)
       AND (#modbusInterface."Register Address" = #address)
       AND (#modbusInterface.Mode = 1))
       )
   THEN
       IF (#modbusInterface.Done) THEN
           //Inspect type of output and set correct type of input in modbus register
           #status := #WRITE_OK;
           #modbusInterface.locked := FALSE;
       END_IF;
       IF (#modbusInterface.Error) THEN
           #status := #modbusInterface.Status;
           #modbusInterface.locked := false;
       END_IF;
   END_IF;
END_FUNCTION

FUNCTION "ModbusPollingDelay" : Void   // FC895, SCL
TITLE = ModbusPollingDelay
{ S7_Optimized_Access := 'TRUE' }
AUTHOR : Matt_Paulissen
FAMILY : AWCModbus
NAME : ModbusPollingDelay
VERSION : 0.1
// The polling delay function is designed to slow down the polling engine in the event it overwhelms a slave or client device.  A delay time is given and all blocks below the polling delay won’t be called until into the time entered into Delay Time elapses.
   VAR_INPUT
      timerID : Int;   // This must be a unique number for every polling delay block that is called in the user program.
      delayTime : Time;   // The amount of time the block will delay the next Modbus polling function.
   END_VAR
   VAR_IN_OUT
      modbusInterface : "typeMasterData";   // The “Master Interface” parameter is used to pass date between the Modbus RTU Engine and subsequent read and write function. The data type is the user defined type “typeMasterData”. It is necessary to create a global data block containing one instance of the “typeMasterData”.
   END_VAR
   VAR_TEMP
      tempPosition : DInt;
      tempStatus : Int;
      tempCurrentTime : DTL;
      tempStartTime : DTL;
      tempEndTime : DTL;
   END_VAR
BEGIN
   REGION BLOCK INFO HEADER
       //===============================================================================
       // AWC INC / (c)Copyright 2022
       //-------------------------------------------------------------------------------
       // Title:            ModbusPollingDelay_xxx
       // Comment/Function: Delay Polling Group
       // Library/Family:   AWCModbus
       // Author:           Matt Paulissen
       // Tested with:      ---
       // Engineering:      TIA Portal V17
       // Restrictions:     ---
       // Requirements:     ---
       //-------------------------------------------------------------------------------
       // Change log table:
       // Version  | Date       | Expert in charge       | Changes applied
       //----------|------------|------------------------|------------------------------
       // 01.00.00 | 01.08.2019 | Matt Paulissen | First released version
       //===============================================================================
   END_REGION

   REGION DESCRIPTION
       (/*The polling delay function is designed to slow down the polling engine in the event it overwhelms a slave or client device.
       A delay time is given and all blocks below the polling delay won’t be called until into the time entered into Delay Time elapses.*/)
   END_REGION DESCRIPTION

   //Check for lock
   IF (NOT #modbusInterface.locked) THEN
       //Create ID out of current PLC time
       #tempStatus := RD_SYS_T(#tempCurrentTime);
       //Serialize start time into interface
       #tempPosition := 0;
       #tempStatus := Serialize(SRC_VARIABLE := #tempCurrentTime, DEST_ARRAY => #modbusInterface.Data, POS := #tempPosition);
       #modbusInterface."Slave ID" := 0;
       #modbusInterface."Register Address" := #timerID;
       #modbusInterface.Mode := 0;
       #modbusInterface.Length := 0;
       #modbusInterface.locked := TRUE;
       #modbusInterface.RequestID += 1;
       RETURN;
   END_IF;
   IF ((#modbusInterface.locked)
       AND (
       (#modbusInterface."Slave ID" = 0)
       AND (#modbusInterface."Register Address" = #timerID)
       AND (#modbusInterface.Mode = 0))
       )
   THEN
       #tempPosition := 0;
       #tempStatus := Deserialize(SRC_ARRAY := #modbusInterface.Data, DEST_VARIABLE => #tempStartTime, POS := #tempPosition);
       #tempEndTime := T_ADD(IN1 := #tempStartTime, IN2 := #delayTime);
       #tempStatus := RD_SYS_T(#tempCurrentTime);
       IF (#tempCurrentTime > #tempEndTime) THEN
           #modbusInterface.locked := FALSE;
       END_IF;
   END_IF;
END_FUNCTION

// folder: AWCModbus/02_Modbus Devices/Cameron

FUNCTION "NuFlo" : Void   // FC897, SCL
TITLE = NuFlo
{ S7_Optimized_Access := 'TRUE' }
AUTHOR : Matt_Paulissen
FAMILY : AWCModbus
NAME : NuFlo
VERSION : 0.1
// The NuFlo function block is used to poll Cameron NuFlo flow meters
   VAR_INPUT
      slaveId : Int;   // When using the function for Modbus RTU this will be the remote slave network address. When using the function for Modbus TCP this will be the device address, in most instances this value will be 1, unless there is a Modbus TCP to Modbus RTU gateway employed. If there is a Modbus TCP to Modbus RTU gateway this value will point to the slave device address on the Modbus RTU side of the gateway.
   END_VAR
   VAR_OUTPUT
      currentFlow : Variant;   // Current flow from transmitter
      currentTotal : Variant;   // Current totalizer value from transmitter
      grandTotal : Variant;   // Current grand total from totalizer
   END_VAR
   VAR_IN_OUT
      modbusInterface : "typeMasterData";   // The “Master Interface” parameter is used to pass date between the Modbus RTU Engine and subsequent read and write function. The data type is the user defined type “typeMasterData”. It is necessary to create a global data block containing one instance of the “typeMasterData”.
   END_VAR
BEGIN
   REGION BLOCK INFO HEADER
       //===============================================================================
       // AWC INC / (c)Copyright 2022
       //-------------------------------------------------------------------------------
       // Title:            NuFlo_xxx
       // Comment/Function: Read data from Cameron NuFlu Flowmeter
       // Library/Family:   AWCModbus
       // Author:           Matt Paulissen
       // Tested with:      ---
       // Engineering:      TIA Portal V17
       // Restrictions:     ---
       // Requirements:     ---
       //-------------------------------------------------------------------------------
       // Change log table:
       // Version  | Date       | Expert in charge       | Changes applied
       //----------|------------|------------------------|------------------------------
       // 01.00.00 | 01.08.2019 | Matt Paulissen | First released version
       // 01.00.01 | 11.16.2022 | Matt Paulissen | Updated General Poll
       //===============================================================================
   END_REGION

   REGION DESCRIPTION
       (/*The NuFlo function block is used to poll Cameron NuFlo flow meters.*/)
   END_REGION DESCRIPTION

   //Current Flow
   "GeneralModbusPoll"(slaveId:=#slaveId,
                       address:=48013,
                       swappedFloatingPoint:=false,
                       substituteValue:=0.0,
                       data=>#currentFlow,
                       modbusInterface:=#modbusInterface);
   //Current Total
   "GeneralModbusPoll"(slaveId := #slaveId,
                       address := 48027,
                       swappedFloatingPoint := false,
                       substituteValue := 0.0,
                       data => #currentTotal,
                       modbusInterface := #modbusInterface);
   //Grand Total
   "GeneralModbusPoll"(slaveId := #slaveId,
                       address := 48011,
                       swappedFloatingPoint := false,
                       substituteValue := 0.0,
                       data => #grandTotal,
                       modbusInterface := #modbusInterface);
END_FUNCTION

// folder: AWCModbus/02_Modbus Devices/ElectroLab

FUNCTION "LevelStick2100" : Void   // FC898, SCL
TITLE = LevelStick2100
{ S7_Optimized_Access := 'TRUE' }
AUTHOR : Matt_Paulissen
FAMILY : AWCModbus
NAME : LevelStick2100
VERSION : 0.1
// The ElectroLab 2100 block is used to poll 2100 level sticks.  The block will get the level and interface level in inches * 100.
   VAR_INPUT
      slaveId : Int;   // When using the function for Modbus RTU this will be the remote slave network address. When using the function for Modbus TCP this will be the device address, in most instances this value will be 1, unless there is a Modbus TCP to Modbus RTU gateway employed. If there is a Modbus TCP to Modbus RTU gateway this value will point to the slave device address on the Modbus RTU side of the gateway.
   END_VAR
   VAR_OUTPUT
      level : Variant;   // Current level in inches * 100
      interfaceLevel : Variant;   // Current interface level in inches * 100
   END_VAR
   VAR_IN_OUT
      modbusInterface : "typeMasterData";   // The “Master Interface” parameter is used to pass date between the Modbus RTU Engine and subsequent read and write function. The data type is the user defined type “typeMasterData”. It is necessary to create a global data block containing one instance of the “typeMasterData”.
   END_VAR
BEGIN
   REGION BLOCK INFO HEADER
       //===============================================================================
       // AWC INC / (c)Copyright 2022
       //-------------------------------------------------------------------------------
       // Title:            LevelStick2100_xxx
       // Comment/Function: Read data from Cameron NuFlu Flowmeter
       // Library/Family:   AWCModbus
       // Author:           Matt Paulissen
       // Tested with:      ---
       // Engineering:      TIA Portal V17
       // Restrictions:     ---
       // Requirements:     ---
       //-------------------------------------------------------------------------------
       // Change log table:
       // Version  | Date       | Expert in charge       | Changes applied
       //----------|------------|------------------------|------------------------------
       // 01.00.00 | 01.08.2019 | Matt Paulissen | First released version
       // 01.00.01 | 11.16.2022 | Matt Paulissen | Updated General Poll
       //===============================================================================
   END_REGION

   REGION DESCRIPTION
       (/*The ElectroLab 2100 block is used to poll 2100 level sticks. The block will get the level and interface $\text{level in inches} \times 100$.*/)
   END_REGION DESCRIPTION

   //Current Velocity
   "GeneralModbusPoll"(slaveId:=#slaveId,
                       address:=43991,
                       swappedFloatingPoint:=false,
                       substituteValue:=0.0,
                       data=>#level,
                       modbusInterface:=#modbusInterface);
   "GeneralModbusPoll"(slaveId := #slaveId,
                       address := 43992,
                       swappedFloatingPoint := false,
                       substituteValue := 0.0,
                       data => #interfaceLevel,
                       modbusInterface := #modbusInterface);
END_FUNCTION

// folder: AWCModbus/02_Modbus Devices/Siemens

FUNCTION "Mag6or8000" : Void   // FC896, SCL
TITLE = Mag6or8000
{ S7_Optimized_Access := 'TRUE' }
AUTHOR : Matt_Paulissen
FAMILY : AWCModbus
NAME : Mag6or8000
VERSION : 0.1
// This block will poll Siemens Mag 6000 or 8000 flow meters and return velocity, flow, and totalizer readings.
   VAR_INPUT
      slaveId : Int;   // When using the function for Modbus RTU this will be the remote slave network address. When using the function for Modbus TCP this will be the device address, in most instances this value will be 1, unless there is a Modbus TCP to Modbus RTU gateway employed. If there is a Modbus TCP to Modbus RTU gateway this value will point to the slave device address on the Modbus RTU side of the gateway.
   END_VAR
   VAR_OUTPUT
      velocity : Variant;   // Current flow from transmitter
      flow : Variant;   // Current totalizer value from transmitter
      totalizer : Variant;   // Current total from totalizer
   END_VAR
   VAR_IN_OUT
      modbusInterface : "typeMasterData";   // The “Master Interface” parameter is used to pass date between the Modbus RTU Engine and subsequent read and write function. The data type is the user defined type “typeMasterData”. It is necessary to create a global data block containing one instance of the “typeMasterData”.
   END_VAR
   VAR_TEMP
      tempStatus : Int;
   END_VAR
BEGIN
   REGION BLOCK INFO HEADER
       //===============================================================================
       // AWC INC / (c)Copyright 2022
       //-------------------------------------------------------------------------------
       // Title:            Mag6or8000_xxx
       // Comment/Function: Read values from Siemens Mag Meters
       // Library/Family:   AWCModbus
       // Author:           Matt Paulissen
       // Tested with:      ---
       // Engineering:      TIA Portal V17
       // Restrictions:     ---
       // Requirements:     ---
       //-------------------------------------------------------------------------------
       // Change log table:
       // Version  | Date       | Expert in charge       | Changes applied
       //----------|------------|------------------------|------------------------------
       // 01.00.00 | 01.14.2019 | Matt Paulissen | First released version
       // 01.00.01 | 11.16.2022 | Matt Paulissen | Updated General Poll
       //===============================================================================
   END_REGION

   REGION DESCRIPTION
       (/*This block will poll Siemens Mag 6000 or 8000 flow meters and return velocity, flow, and totalizer readings.*/)
   END_REGION DESCRIPTION

   //Current Velocity
   "GeneralModbusPoll"(slaveId:=#slaveId,
                       address:=42999,
                       swappedFloatingPoint:=false,
                       substituteValue:=0.0,
                       data=>#velocity,
                       modbusInterface:=#modbusInterface);
   //Current Flow
   "GeneralModbusPoll"(slaveId := #slaveId,
                       address := 43001,
                       swappedFloatingPoint := false,
                       substituteValue := 0.0,
                       data => #flow,
                       modbusInterface := #modbusInterface);
   //Totalizer
   "LargeModbusPoll"(slaveId:=#slaveId,
                     address:=43016
                     ,
                     data=>#totalizer,
                     status=> #tempStatus,
                     modbusInterface:=#modbusInterface);
END_FUNCTION

// folder: AWCModbus/02_Modbus Devices/Tosibox

FUNCTION_BLOCK "PollTosibox"   // FB1, SCL
{ S7_Optimized_Access := 'TRUE' }
VERSION : 0.1
   VAR_INPUT
      slaveId : Int;   // modbus slave id
   END_VAR
   VAR_OUTPUT
      latitude : LReal;
      longitude : LReal;
      UTCTime : LReal;
   END_VAR
   VAR_IN_OUT
      modbusInterface : "typeMasterData";
   END_VAR
   VAR
      statData : Array[0..11] of Int;
      statLat : Array[0..7] of Byte;
      statLon : Array[0..7] of Byte;
      statUTC : Array[0..7] of Byte;
   END_VAR
   VAR_TEMP
      tempStatus : Int;
      tempPos : DInt;
   END_VAR
BEGIN
   REGION BLOCK INFO HEADER
       //===============================================================================
       // AWC INC / (c)Copyright 2022
       //-------------------------------------------------------------------------------
       // Title:            PollTosibox_xxx
       // Comment/Function: Get Modbus Values from TosiMox
       // Library/Family:   AWCModbus
       // Author:           Matt Paulissen
       // Tested with:      ---
       // Engineering:      TIA Portal V17
       // Restrictions:     ---
       // Requirements:     ---
       //-------------------------------------------------------------------------------
       // Change log table:
       // Version  | Date       | Expert in charge       | Changes applied
       //----------|------------|------------------------|------------------------------
       // 01.00.00 | 07.30.2020 | Matt Paulissen | First released version
       // 01.00.01 | 11.16.2022 | Matt Paulissen | Updated General Poll
       //===============================================================================
   END_REGION

   REGION DESCRIPTION
       (/*This block will poll Tosibox Image on Moxa for GPS and Time.*/)
   END_REGION DESCRIPTION
   "LargeModbusPoll"(slaveId:=1,
                     address:=40001,
                     data=>#statData,
                     status=>#tempStatus,
                     modbusInterface:=#modbusInterface);
   //Parse Latitude
   #statLat[0] := #statData[3].%B1;
   #statLat[1] := #statData[3].%B0;
   #statLat[2] := #statData[2].%B1;
   #statLat[3] := #statData[2].%B0;
   #statLat[4] := #statData[1].%B1;
   #statLat[5] := #statData[1].%B0;
   #statLat[6] := #statData[0].%B1;
   #statLat[7] := #statData[0].%B0;

   #tempPos := 0;
   #tempStatus := Deserialize(SRC_ARRAY := #statLat, DEST_VARIABLE => #latitude, POS := #tempPos);
   //Parse Longitude
   #statLon[0] := #statData[7].%B1;
   #statLon[1] := #statData[7].%B0;
   #statLon[2] := #statData[6].%B1;
   #statLon[3] := #statData[6].%B0;
   #statLon[4] := #statData[5].%B1;
   #statLon[5] := #statData[5].%B0;
   #statLon[6] := #statData[4].%B1;
   #statLon[7] := #statData[4].%B0;

   #tempPos := 0;
   #tempStatus := Deserialize(SRC_ARRAY := #statLon, DEST_VARIABLE => #longitude, POS := #tempPos);

   //Parse Time
   #statUTC[0] := #statData[11].%B1;
   #statUTC[1] := #statData[11].%B0;
   #statUTC[2] := #statData[10].%B1;
   #statUTC[3] := #statData[10].%B0;
   #statUTC[4] := #statData[9].%B1;
   #statUTC[5] := #statData[9].%B0;
   #statUTC[6] := #statData[8].%B1;
   #statUTC[7] := #statData[8].%B0;

   #tempPos := 0;
   #tempStatus := Deserialize(SRC_ARRAY := #statUTC, DEST_VARIABLE => #UTCTime, POS := #tempPos);
END_FUNCTION_BLOCK